SUBAPPLICATION Uebung_011c (* Numeric Value Input I3 Durchschleifen auf N3 *)
  (* Standard: 61499-2; Description: Copyright (c) 2023 Meisterschulen am Ostbahnhof This program and the accompanying materials are made available under the terms of the Eclipse Public License 2.0 which is available at https://www.eclipse.org/legal/epl-2.0/ SPDX-License-Identifier: EPL-2.0 *)
  (* Version 1.0, 2026-04-14, Franz Höpfinger, Meisterschulen am Ostbahnhof, initial API and implementation and/or initial documentation *)
  PACKAGE Uebungen;
  IMPORT Uebungen::const::UT::DefaultPool::InputNumber_I3;
  IMPORT Uebungen::const::UT::DefaultPool::OutputNumber_N3;
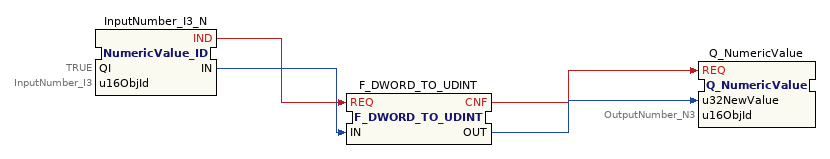
  FBS
    InputNumber_I3_N : isobus::UT::io::NumericValue::NumericValue_ID(QI := TRUE, u16ObjId := InputNumber_I3);
    F_DWORD_TO_UDINT : iec61131::conversion::F_DWORD_TO_UDINT;
    Q_NumericValue : isobus::UT::Q::Q_NumericValue(u16ObjId := OutputNumber_N3);
  END_FBS
  EVENT_CONNECTIONS
    F_DWORD_TO_UDINT.CNF TO Q_NumericValue.REQ;
    InputNumber_I3_N.IND TO F_DWORD_TO_UDINT.REQ;
  END_CONNECTIONS
  DATA_CONNECTIONS
    F_DWORD_TO_UDINT.OUT TO Q_NumericValue.u32NewValue;
    InputNumber_I3_N.IN TO F_DWORD_TO_UDINT.IN;
  END_CONNECTIONS
END_SUBAPPLICATION
